// TIA Portal project "Projekt_PLC_Kwiatkowski_V18" (V18)

(* hardware
DEVICE "S7-1200 station_1"  S7-1200 Station
   slot 0: "Rack_0"  S7-1200 Rack  Rack  V1.0
   slot 1: "PLC_1"  CPU 1214C DC/DC/DC  6ES7 214-1AG40-0XB0  V4.2
      slot 3: "AQ 1x12BIT_1"  AQ1 signal board  6ES7 232-4HA30-0XB0  V1.0
*)

// ===== PLC "PLC_1"  CPU 1214C DC/DC/DC =====

VAR_GLOBAL   // PLC tag table "Default tag table"
   "tagStart" AT %I0.0 : Bool;
   "tagStop" AT %I0.1 : Bool;
   "tagReset" AT %I0.2 : Bool;
   "tagLampRun" AT %Q0.0 : Bool;
   "tagLampStop" AT %Q0.1 : Bool;
   "tagLampAlarm" AT %Q0.2 : Bool;
   "tagLevelRaw" AT %IW30 : Int;
   "tagFillValve" AT %QW64 : Int;
   "tagDrainValve" AT %QW66 : Int;
END_VAR

DATA_BLOCK "FbTankBatch_DB"   // DB1
{ S7_Optimized_Access := 'TRUE' }
VERSION : 0.1
// stored: InstanceOfName FbTankBatch
"FbTankBatch"
BEGIN
   statSetpoint := 60.0;
END_DATA_BLOCK

FUNCTION_BLOCK "FbTankBatch"   // FB1, SCL
{ S7_Optimized_Access := 'TRUE' }
VERSION : 0.1
// ------------------------------------------------------------------------------
//  BLOK FUNKCYJNY: sterowanie wsadowe (napelnianie -> przetrzymanie -> spust)
// ------------------------------------------------------------------------------
   VAR_INPUT
      start : Bool;   // przycisk Start (Factory I/O)
      stop : Bool;   // przycisk Stop
      reset : Bool;   // przycisk Reset
      levelRaw : Int;   // Level Meter - surowa wartosc analogowa
   END_VAR
   VAR_OUTPUT
      fillValve : Int;   // Fill Valve - analogowe wyjscie 0..RAW_MAX
      drainValve : Int;   // Discharge Valve - analogowe wyjscie 0..RAW_MAX
      lampRun : Bool;   // lampka pracy
      lampStop : Bool;   // lampka stanu spoczynku
      lampAlarm : Bool;   // lampka alarmu zmienne statyczne
   END_VAR
   VAR
      statState : Int;   // stan maszyny: 0..5
      statLevelPct : Real;   // przefiltrowany poziom [%]
      statSetpoint : Real := 55.0;   // zadany poziom [%] - edytowalny online
      statBatchCount : Int;   // liczba ukonczonych wsadow
      statSampleIdx : Int;   // indeks bufora filtra
      statSamples : Array[0..4] of Real;   // bufor probek do sredniej kroczacej
      instStartEdge : R_TRIG;   // detekcja zbocza przycisku Start
      instStopEdge : R_TRIG;   // detekcja zbocza przycisku Stop
      instFillTon : TON_TIME;   // watchdog czasu napelniania
      instHoldTon : TON_TIME;   // czas przetrzymania / mieszania
      instBatchCtu : CTU_INT;   // licznik wsadow
   END_VAR
   VAR RETAIN
      instDrainTon : TON_TIME;
   END_VAR
   VAR_TEMP
      tempStartPulse : Bool;
      tempStopPulse : Bool;
      tempFillTimeout : Bool;
      tempHoldDone : Bool;
      tempAllDone : Bool;
      tempRunning : Bool;
      tempI : Int;
      tempSum : Real;
      tempErr : Real;
      tempCmd : Real;
      tempDrainDone : Bool;
   END_VAR
   VAR CONSTANT
      KP : Real := 8.0;   // wzmocnienie czlonu P
      RAW_MAX : Int := 27648;   // pelna skala analogu (Siemens)
      LEVEL_MAX : Real := 100.0;   // gorny zakres poziomu [%]
      SAMPLE_COUNT : Int := 5;   // liczba probek filtra
      FILL_TIMEOUT : Time := T#30S;   // limit czasu napelniania
      HOLD_TIME : Time := T#5S;   // czas przetrzymania
      BATCH_TARGET : Int := 3;   // ile wsadow ma wykonac
      EMPTY_LEVEL : Real := 2.0;   // prog "zbiornik pusty" [%]
      DRAIN_HOLD : Time := T#4S;
   END_VAR
BEGIN
       // 1) DETEKCJA ZBOCZY na przyciskach Start / Stop
       // 
       #instStartEdge(CLK := #start);
       #tempStartPulse := #instStartEdge.Q;
       #instStopEdge(CLK := #stop);
       #tempStopPulse := #instStopEdge.Q;


       // 2) SYGNAL ANALOGOWY: skalowanie (FC z NORM_X/SCALE_X) i zapis do bufora

       #statSamples[#statSampleIdx] := "FcScaleLevel"(rawValue := #levelRaw,
                                                      rawMax := #RAW_MAX,
                                                      engMax := #LEVEL_MAX);
       #statSampleIdx := #statSampleIdx + 1;
       IF #statSampleIdx >= #SAMPLE_COUNT THEN
           #statSampleIdx := 0;
       END_IF;


       // 3) PETLA FOR - srednia kroczaca (z instrukcjami CONTINUE oraz EXIT)

       #tempSum := 0.0;
       FOR #tempI := 0 TO #SAMPLE_COUNT - 1 DO
           IF #statSamples[#tempI] < 0.0 THEN
               CONTINUE;                  // pomin bledna probke, petla trwa dalej
           END_IF;
           IF #statSamples[#tempI] > 200.0 THEN
               EXIT;                      // wartosc uszkodzona - przerwij petle
           END_IF;
           #tempSum := #tempSum + #statSamples[#tempI];
       END_FOR;
       #statLevelPct := #tempSum / INT_TO_REAL(#SAMPLE_COUNT);


       // 4) TIMERY - wolane co cykl, wejscie IN zwiazane ze stanem (auto-reset)

       #instFillTon(IN := (#statState = 1),
                    PT := #FILL_TIMEOUT);
       #tempFillTimeout := #instFillTon.Q;
       #instHoldTon(IN := (#statState = 2),
                    PT := #HOLD_TIME);
       #tempHoldDone := #instHoldTon.Q;
       #instDrainTon(IN := (#statState = 3) AND (#statLevelPct <= #EMPTY_LEVEL),
                     PT := #DRAIN_HOLD);
       #tempDrainDone := #instDrainTon.Q;

       // 5) LICZNIK wsadow - zlicza wejscie w stan 4 (koniec wsadu)

       #instBatchCtu(CU := (#statState = 4),
                     R := #reset,
                     PV := #BATCH_TARGET);
       #statBatchCount := #instBatchCtu.CV;
       #tempAllDone := (#statBatchCount >= #BATCH_TARGET);


       // 6) STOP / RESET - nadrzedne (logika + zbocza + petla WHILE)

       IF #tempStopPulse THEN
           #statState := 0;
       END_IF;
       IF #reset THEN
           #statState := 0;
           #tempI := 0;
           WHILE #tempI < #SAMPLE_COUNT DO  
               #statSamples[#tempI] := 0.0;
               #tempI := #tempI + 1;
           END_WHILE;
       END_IF;


       // 7) MASZYNA STANOW (CASE) - sekwencja wsadowa

       CASE #statState OF
           0:  // IDLE - oczekiwanie na Start
               #fillValve := 0;
               #drainValve := 0;
               IF #tempStartPulse THEN
                   #statState := 1;
               END_IF;

           1:  // FILLING - proporcjonalne otwarcie zaworu (sterowanie analogowe)
               #drainValve := 0;
               #tempErr := #statSetpoint - #statLevelPct;   // arytmetyka: uchyb
               #tempCmd := #tempErr * #KP;                   // czlon proporcjonalny
               IF #tempCmd > 100.0 THEN                      // ograniczenie wyjscia
                   #tempCmd := 100.0;
               ELSIF #tempCmd < 50.0 THEN
                   #tempCmd := 50.0;
               END_IF;
               // procent -> surowa wartosc analogowa
               #fillValve := REAL_TO_INT(#tempCmd / 100.0 * INT_TO_REAL(#RAW_MAX));
               IF #statLevelPct >= #statSetpoint THEN
                   #statState := 2;
               ELSIF #tempFillTimeout THEN
                   #statState := 5;                           // przekroczony czas -> ALARM
               END_IF;

           2:  // HOLDING - przetrzymanie / mieszanie
               #fillValve := 0;
               #drainValve := 0;
               IF #tempHoldDone THEN
                   #statState := 3;
               END_IF;

           3:  // DRAINING - oproznianie
               #fillValve := 0;
               #drainValve := #RAW_MAX;
              IF #tempDrainDone THEN
                   #statState := 4;
               END_IF;

           4:  // BATCH DONE - kolejny wsad czy koniec
               #drainValve := 0;
               IF #statBatchCount >= #BATCH_TARGET THEN
                   #statState := 0;                           // wszystkie wsady gotowe
               ELSE
                   #statState := 1;                           // start kolejnego wsadu
               END_IF;

           ELSE:  // 5 = ALARM oraz kazdy inny nieoczekiwany stan (wymog Styleguide)
               #fillValve := 0;
               #drainValve := 0;
       END_CASE;


       // 8) SYGNALIZACJA - funkcje logiczne (AND / OR / NOT)

       #tempRunning := (#statState = 1) OR (#statState = 2) OR (#statState = 3);
       #lampRun := #tempRunning AND NOT #tempAllDone;
       #lampStop := (#statState = 0);
       #lampAlarm := (#statState = 5);
END_FUNCTION_BLOCK

FUNCTION "FcScaleLevel" : Real   // FC1, SCL
{ S7_Optimized_Access := 'TRUE' }
VERSION : 0.1
// ==============================================================================
//  Projekt zaliczeniowy - Zaawansowane PLC (SCL)
//  Sterowanie wsadowe zbiornikiem (Factory I/O: scena "Level Control")
//  Plik zrodlowy do importu: External source files -> Generate blocks from source
// 
//  Zawiera:
//    FC "FcScaleLevel"  - skalowanie sygnalu analogowego (NORM_X / SCALE_X, RETURN)
//    FB "FbTankBatch"   - logika sekwencji wsadowej (maszyna stanow)
// 
//  Zgodnie z zaleceniami Siemens Styleguide:
//    - identyfikatory camelCase, bez polskich znakow, do 24 znakow
//    - stale WIELKIMI LITERAMI, instancje z prefiksem "inst"
//    - zmienne statyczne "stat", tymczasowe "temp"
// ==============================================================================
// ------------------------------------------------------------------------------
//  FUNKCJA POMOCNICZA: surowa wartosc analogowa -> jednostki inzynierskie [%]
// ------------------------------------------------------------------------------
   VAR_INPUT
      rawValue : Int;   // surowa wartosc z wejscia analogowego (WORD/Int)
      rawMax : Int;   // zakres pelnej skali (np. 27648)
      engMax : Real;   // gorny zakres inzynierski (np. 100.0 %)
   END_VAR
   VAR_TEMP
      tempNorm : Real;   // wartosc znormalizowana 0.0 .. 1.0
   END_VAR
BEGIN
       // Straz wejscia - jesli konfiguracja bledna, przerwij funkcje (RETURN)
       IF #rawMax <= 0 THEN
           #FcScaleLevel := 0.0;
           RETURN;
       END_IF;

       // Normalizacja surowej wartosci do zakresu 0.0 .. 1.0
       #tempNorm := NORM_X(MIN := 0, MAX := #rawMax, VALUE := #rawValue);

       // Skalowanie do jednostek inzynierskich (procenty)
       #FcScaleLevel := SCALE_X(MIN := 0.0, MAX := #engMax, VALUE := #tempNorm);
END_FUNCTION

ORGANIZATION_BLOCK "Main"   // OB1, LAD, ProgramCycle
TITLE = "Main Program Sweep (Cycle)"
{ S7_Optimized_Access := 'TRUE' }
VERSION : 0.1
   VAR_INPUT
      Initial_Call : Bool;   // Initial call of this OB
      Remanence : Bool;   // =True, if remanent data are available
   END_VAR
BEGIN

REGION Network 1 (SCL)
   // Main [OB1] w SCL — wywolanie bloku sterowania wsadowego

   "FbTankBatch_DB"(start := "tagStart",
                    stop := "tagStop",     
                    reset := "tagReset",
                    levelRaw := "tagLevelRaw",
                    fillValve => "tagFillValve",
                    drainValve => "tagDrainValve",
                    lampRun => "tagLampRun",
                    lampStop => "tagLampStop",
                    lampAlarm => "tagLampAlarm");
END_REGION
END_ORGANIZATION_BLOCK